PROGRAM AxisRotate
VAR_INPUT
	Desired_Speed: INT ;
	Desired_Position: UINT ;
	tolerance: UINT;
END_VAR
VAR
	Axis : ST_Axis := (
		uiCounterValue := INPUT.IW_VGR_CounterValueRotate,
		bSetCounter := OUTPUT.QX_VGR_SetCounterRotate,
		uiSetCounterValue := OUTPUT.QW_VGR_SetCounterValueRotate,
		iControl := VGR.QW_VGR_PWM_Rotate_Control,
		iPWM := VGR.QW_VGR_PWM_Rotate_M3,
		bJogMinus := VGR.QX_VGR_M3_RotateClockwise_Q5,
		bJogPlus := VGR.QX_VGR_M3_RotateCounterclockwise_Q6
	);
	Motor_Direction_Rotational: Motor_direction;
END_VAR

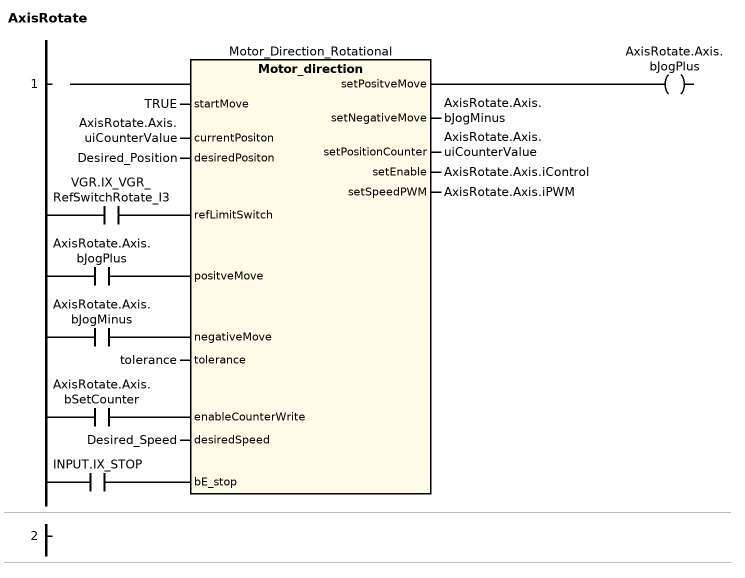
// NETWORK 1
Motor_Direction_Rotational(
    startMove := TRUE,
    currentPositon := AxisRotate.Axis.uiCounterValue,
    desiredPositon := Desired_Position,
    refLimitSwitch := VGR.IX_VGR_RefSwitchRotate_I3,
    positveMove := AxisRotate.Axis.bJogPlus,
    negativeMove := AxisRotate.Axis.bJogMinus,
    tolerance := tolerance,
    enableCounterWrite := AxisRotate.Axis.bSetCounter,
    desiredSpeed := Desired_Speed,
    bE_stop := INPUT.IX_STOP,
    setNegativeMove => AxisRotate.Axis.bJogMinus,
    setPositionCounter => AxisRotate.Axis.uiCounterValue,
    setEnable => AxisRotate.Axis.iControl,
    setSpeedPWM => AxisRotate.Axis.iPWM); // Motor_direction
AxisRotate.Axis.bJogPlus := Motor_Direction_Rotational.setPositveMove;

// NETWORK 2

END_PROGRAM

(* stored: Version 1.1.0.1, ProductVersion 3.1.4024.12
   POU AxisRotate: Id {983dc9d9-cdec-4c33-92b3-8daef21be09c}, SpecialFunc None *)
